PROGRAM MAIN
VAR
END_VAR

END_PROGRAM

(* stored: Version 1.1.0.1
   POU MAIN: Id {473e1599-14d9-4e95-b23a-b4efec4cea01} *)
